FUNCTION_BLOCK PUBLIC FB_JednorazowyBoolin
VAR
	_boolin : BOOL;	
END_VAR

PROPERTY PUBLIC boolin : BOOL
GET
boolin := _boolin;
END_GET
SET
_boolin := boolin;
END_SET
END_PROPERTY

END_FUNCTION_BLOCK

(* stored: Version 1.1.0.1
   POU FB_JednorazowyBoolin: Id {356d8125-8fe1-078d-20b2-469f11cd746b}, SpecialFunc None
   Property boolin: Id {98cbbf20-9582-01e7-042a-c965b007bd8b}
   Get Get: Id {72345106-28a3-00da-1829-e1ed8abe2fcf}
   Set Set: Id {f2aed263-f562-0b2f-1362-c51dee4ea99e} *)
